FUNCTION_BLOCK FB_Sensor
VAR_INPUT
END_VAR
VAR_OUTPUT
END_VAR
VAR
	{attribute 'OPC.UA.DA' := '1'}
	bSignal  AT%I* : BOOL;	
END_VAR

PROPERTY GetSignal : BOOL
GET
GetSignal := bSignal;
END_GET
END_PROPERTY

END_FUNCTION_BLOCK

(* stored: Version 1.1.0.1, ProductVersion 3.1.4022.12
   POU FB_Sensor: Id {5cdbb8eb-2ee3-4428-8e06-45109b7bda85}, SpecialFunc None
   Property GetSignal: Id {b1873d3f-9164-488f-a0ca-83841b40c1e0}
   Get Get: Id {f31317ee-353f-4159-90ff-cf9d4b984dfb} *)
